{attribute 'qualified_only'}
{attribute 'strict'}
{attribute 'to_string'}
TYPE enProductTypes_1 :
(
	_PSA := 1,
	PORSCHE_992 := 2,
	VOLVO_SPA := 3,
	_8P0 := 4,
	JAGUAR_FGA_TC02_0040 := 0,	// -> 0
	HAOS_FGA_TC01_0006 := 5,	// -> 5
	NISSAN_FGA_TC01_0007:= 6,	// -> 6
	MERCEDES:= 7,				// -> 7
	FGA_TC02_0049 := 8,
	MAZDA := 9,
	SUBARU := 10,
	BC4 := 11
);
END_TYPE

(* stored: Version 1.1.0.1, ProductVersion 3.1.4024.15
   EnumerationTextList enProductTypes_1: Id {4f609857-32fa-46bc-86ec-8f9b7c787e46} *)
